FUNCTION_BLOCK FB_ErrorHandler IMPLEMENTS ITF_ErrorHandlerSubject
VAR_INPUT
END_VAR
VAR_OUTPUT
END_VAR
VAR
	_arStCBMLInfo		: ARRAY [0..100] OF stCBMLInfo;
	arItfDeviceObserver : ARRAY [0..100] OF ITF_Device;
	uiFc				: UINT;
END_VAR

FOR uiFc:=0 TO 100 BY 1 DO
	IF (arItfDeviceObserver[uiFc] <> 0) THEN
		_arStCBMLInfo[uiFc]:= arItfDeviceObserver[uiFc].P_stCBMLInfo;
	END_IF
END_FOR

METHOD AttachDevice : BOOL
VAR_INPUT
	itfDevice 	: ITF_Device;
END_VAR

VAR 
	uiFc 		: UINT;
END_VAR
FOR uiFc:= 0 TO 100 BY 1 DO
	IF (itfDevice <> 0) AND (arItfDeviceObserver[uiFc] = 0) THEN
		arItfDeviceObserver[uiFc] := itfDevice;
		EXIT;
	END_IF
END_FOR
END_METHOD

END_FUNCTION_BLOCK

(* stored: Version 1.1.0.1, ProductVersion 3.1.4024.11
   POU FB_ErrorHandler: Id {104fbfda-2cee-4df9-aac9-1f1d69a87b3a}, SpecialFunc None
   Method AttachDevice: Id {4242671a-1ddb-4a53-9784-fcc12b7c7eb7} *)
